(* Schneider Machine Expert - Basic project es1_2pompe_1max_2soglie_scelta_alternanza, file version 3.0.0.0 *)
(* ProjectInformations: Name=New project *)

HARDWARE
  Cpu 0: TM221C40R
  EthernetConfiguration: NetworkName=M221, IpAllocationMode=FixedAddress, IpAddress=0.0.0.0, SubnetMask=0.0.0.0
  SerialLineConfiguration: Baud=Baud19200, Parity=ParityEven, DataBits=DataBits8, StopBits=StopBits1, PhysicalMedium=PhysicalMediumRs485, TransmissionMode=TransmissionModeModbusRtu, SlaveId=1, Addressing=SlaveAddressing
  MastTask: UsePeriodScanMode=false, PeriodScan=100
  FastTask: Period=255
  CpuBehavior: StartingMode=StartAsPreviousState, AutoSaveRamOnEeprom=true, WatchdogPeriod=250

SYMBOLS  (address, symbol, comment, settings)
  %M0       P1_USABILE
  %M1       P2_USABILE
  %M2       P1_SUPERATO_NUMERO_SEC_LAVORATI
  %M3       P2_SUPERATO_NUMERO_SEC_LAVORATI
  %M4       ORA_E_00  "E' mezzanotte?"
  %M5       ALTERNATO_POMPE_GIORNALIERO
  %S6       SB_TB1S  "Time base of 1 s generated by an internal clock"
  %SW51     SW_RTCHHMM  "RTC Function: contains in BCD HHMM: hour and minute"
  %MW0      PROSSIMA_POMPA_CANDIDATA
  %MW1      STRG_ALTERNANZA_ATTUALE
  %TM0      TIMER_POMPA_1  [Preset=10, Base=OneSecond, IsRetentive=true, IsDynamicPreset=true]
  %C0       CONTATORE_P1_SECONDI_LAVORATI  [Preset=0]
  %C1       CONTATORE_P2_SECONDI_LAVORATI  [Preset=0]
  %I0.0     P1_AUTO
  %I0.1     P1_MOTO
  %I0.2     P1_ANOMALIA
  %I0.3     P2_AUTO
  %I0.4     P2_MOTO
  %I0.5     P2_ANOMALIA
  %I0.6     LVL_MIN
  %I0.7     LVL_MAX
  %Q0.0     P1_CMD
  %Q0.1     P2_CMD
  %Q0.2     ERR_STRG_ALTERNANZA_INVALIDA
  %IW0.0    STRG_ALTERNANZA_INPUT  "0 = avvio; 1 = meno ore; 2 = giornaliera semplice;"  [Type=Type_0_10V, Scope=Scope_Normal, Minimum=0, Maximum=1000]

POU New POU
  (* SectionNumber=1 *)

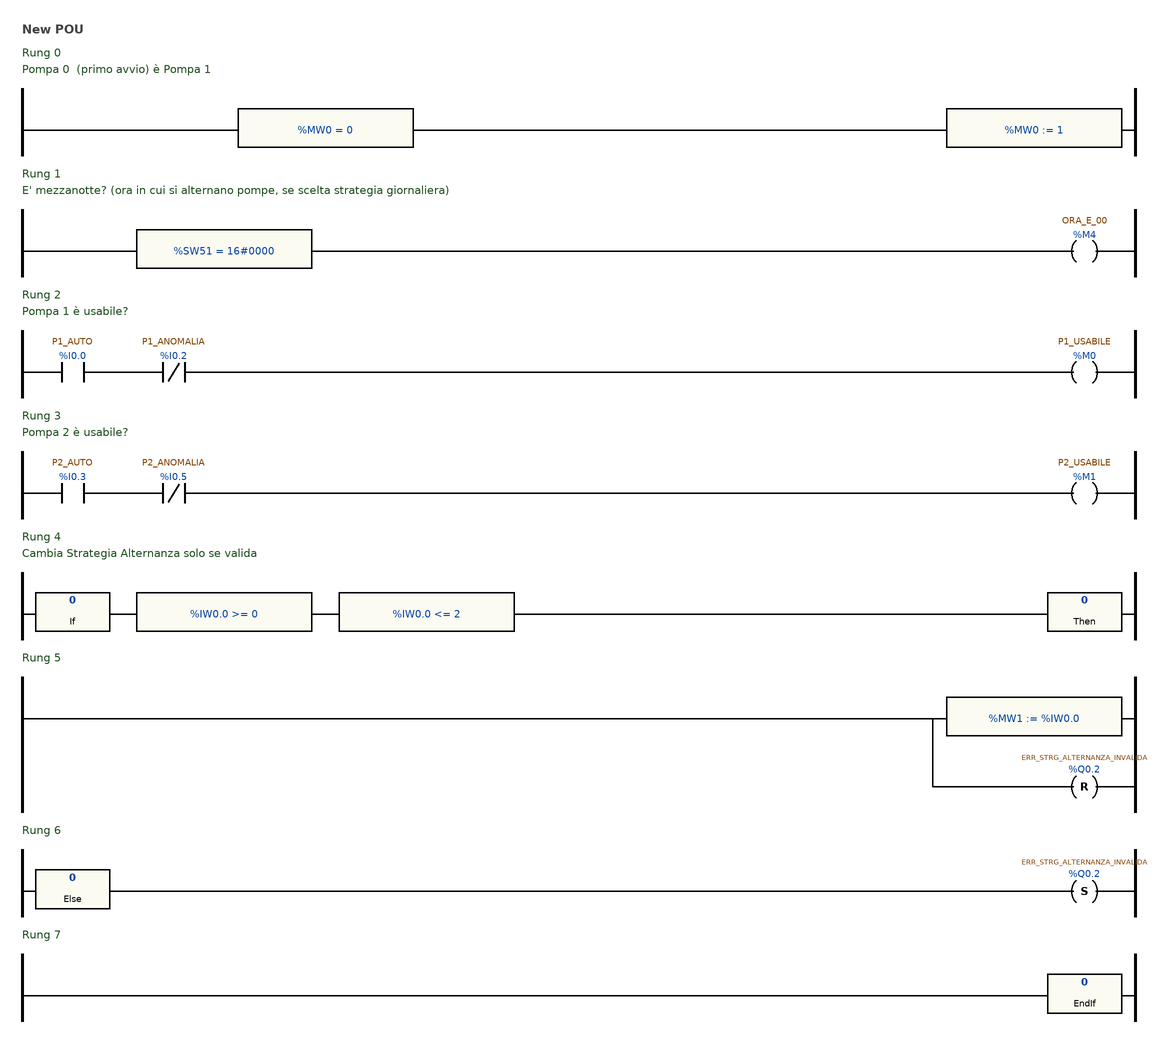

// Rung 0
// Pompa 0  (primo avvio) è Pompa 1
  LD [ %MW0 = 0 ]         (* PROSSIMA_POMPA_CANDIDATA *)
  [ %MW0 := 1 ]           (* PROSSIMA_POMPA_CANDIDATA *)
  // as ST:
  //   IF PROSSIMA_POMPA_CANDIDATA = 0 THEN PROSSIMA_POMPA_CANDIDATA := 1; END_IF;

// Rung 1
// E' mezzanotte? (ora in cui si alternano pompe, se scelta strategia giornaliera)
  LD [ %SW51 = 16#0000 ]  (* SW_RTCHHMM *)
  ST %M4                  (* ORA_E_00 *)
  // as ST:
  //   ORA_E_00 := SW_RTCHHMM = 16#0000;

// Rung 2
// Pompa 1 è usabile?
  LD %I0.0                (* P1_AUTO *)
  ANDN %I0.2              (* P1_ANOMALIA *)
  ST %M0                  (* P1_USABILE *)
  // as ST:
  //   P1_USABILE := P1_AUTO AND NOT P1_ANOMALIA;

// Rung 3
// Pompa 2 è usabile?
  LD %I0.3                (* P2_AUTO *)
  ANDN %I0.5              (* P2_ANOMALIA *)
  ST %M1                  (* P2_USABILE *)
  // as ST:
  //   P2_USABILE := P2_AUTO AND NOT P2_ANOMALIA;

// Rung 4
// Cambia Strategia Alternanza solo se valida
  IF0
  AND [ %IW0.0 >= 0 ]     (* STRG_ALTERNANZA_INPUT *)
  AND [ %IW0.0 <= 2 ]     (* STRG_ALTERNANZA_INPUT *)
  THEN0

// Rung 5
  LD 1
  [ %MW1 := %IW0.0 ]      (* STRG_ALTERNANZA_ATTUALE, STRG_ALTERNANZA_INPUT *)
  R %Q0.2                 (* ERR_STRG_ALTERNANZA_INVALIDA *)
  // as ST:
  //   STRG_ALTERNANZA_ATTUALE := STRG_ALTERNANZA_INPUT;
  //   ERR_STRG_ALTERNANZA_INVALIDA := FALSE;

// Rung 6
  ELSE0
  S %Q0.2                 (* ERR_STRG_ALTERNANZA_INVALIDA *)

// Rung 7
  LD 1
  ENDIF0

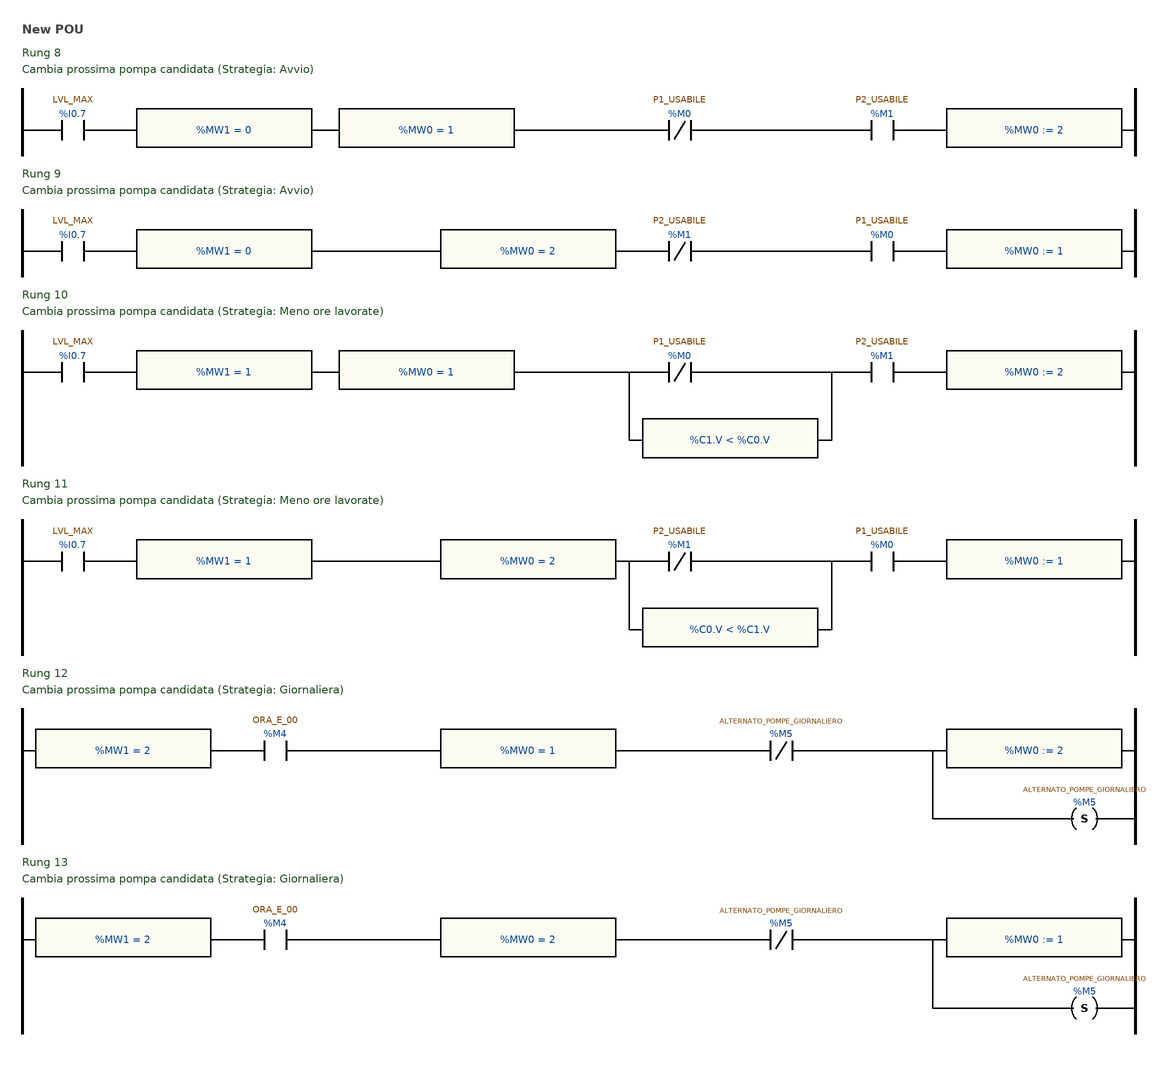

// Rung 8
// Cambia prossima pompa candidata (Strategia: Avvio)
  LD %I0.7                (* LVL_MAX *)
  AND [ %MW1 = 0 ]        (* STRG_ALTERNANZA_ATTUALE *)
  AND [ %MW0 = 1 ]        (* PROSSIMA_POMPA_CANDIDATA *)
  ANDN %M0                (* P1_USABILE *)
  AND %M1                 (* P2_USABILE *)
  [ %MW0 := 2 ]           (* PROSSIMA_POMPA_CANDIDATA *)
  // as ST:
  //   IF LVL_MAX AND STRG_ALTERNANZA_ATTUALE = 0 AND PROSSIMA_POMPA_CANDIDATA = 1 AND NOT P1_USABILE AND P2_USABILE THEN PROSSIMA_POMPA_CANDIDATA := 2; END_IF;

// Rung 9
// Cambia prossima pompa candidata (Strategia: Avvio)
  LD %I0.7                (* LVL_MAX *)
  AND [ %MW1 = 0 ]        (* STRG_ALTERNANZA_ATTUALE *)
  AND [ %MW0 = 2 ]        (* PROSSIMA_POMPA_CANDIDATA *)
  ANDN %M1                (* P2_USABILE *)
  AND %M0                 (* P1_USABILE *)
  [ %MW0 := 1 ]           (* PROSSIMA_POMPA_CANDIDATA *)
  // as ST:
  //   IF LVL_MAX AND STRG_ALTERNANZA_ATTUALE = 0 AND PROSSIMA_POMPA_CANDIDATA = 2 AND NOT P2_USABILE AND P1_USABILE THEN PROSSIMA_POMPA_CANDIDATA := 1; END_IF;

// Rung 10
// Cambia prossima pompa candidata (Strategia: Meno ore lavorate)
  LD %I0.7                (* LVL_MAX *)
  AND [ %MW1 = 1 ]        (* STRG_ALTERNANZA_ATTUALE *)
  AND [ %MW0 = 1 ]        (* PROSSIMA_POMPA_CANDIDATA *)
  AND(N %M0               (* P1_USABILE *)
  OR [ %C1.V < %C0.V ]    (* CONTATORE_P2_SECONDI_LAVORATI, CONTATORE_P1_SECONDI_LAVORATI *)
  )
  AND %M1                 (* P2_USABILE *)
  [ %MW0 := 2 ]           (* PROSSIMA_POMPA_CANDIDATA *)
  // as ST:
  //   IF LVL_MAX AND STRG_ALTERNANZA_ATTUALE = 1 AND PROSSIMA_POMPA_CANDIDATA = 1 AND (NOT P1_USABILE OR CONTATORE_P2_SECONDI_LAVORATI.V < CONTATORE_P1_SECONDI_LAVORATI.V) AND P2_USABILE THEN PROSSIMA_POMPA_CANDIDATA := 2; END_IF;

// Rung 11
// Cambia prossima pompa candidata (Strategia: Meno ore lavorate)
  LD %I0.7                (* LVL_MAX *)
  AND [ %MW1 = 1 ]        (* STRG_ALTERNANZA_ATTUALE *)
  AND [ %MW0 = 2 ]        (* PROSSIMA_POMPA_CANDIDATA *)
  AND(N %M1               (* P2_USABILE *)
  OR [ %C0.V < %C1.V ]    (* CONTATORE_P1_SECONDI_LAVORATI, CONTATORE_P2_SECONDI_LAVORATI *)
  )
  AND %M0                 (* P1_USABILE *)
  [ %MW0 := 1 ]           (* PROSSIMA_POMPA_CANDIDATA *)
  // as ST:
  //   IF LVL_MAX AND STRG_ALTERNANZA_ATTUALE = 1 AND PROSSIMA_POMPA_CANDIDATA = 2 AND (NOT P2_USABILE OR CONTATORE_P1_SECONDI_LAVORATI.V < CONTATORE_P2_SECONDI_LAVORATI.V) AND P1_USABILE THEN PROSSIMA_POMPA_CANDIDATA := 1; END_IF;

// Rung 12
// Cambia prossima pompa candidata (Strategia: Giornaliera)
  LD [ %MW1 = 2 ]         (* STRG_ALTERNANZA_ATTUALE *)
  AND %M4                 (* ORA_E_00 *)
  AND [ %MW0 = 1 ]        (* PROSSIMA_POMPA_CANDIDATA *)
  ANDN %M5                (* ALTERNATO_POMPE_GIORNALIERO *)
  [ %MW0 := 2 ]           (* PROSSIMA_POMPA_CANDIDATA *)
  S %M5                   (* ALTERNATO_POMPE_GIORNALIERO *)
  // as ST:
  //   _t1 := STRG_ALTERNANZA_ATTUALE = 2 AND ORA_E_00 AND PROSSIMA_POMPA_CANDIDATA = 1 AND NOT ALTERNATO_POMPE_GIORNALIERO;
  //   IF _t1 THEN PROSSIMA_POMPA_CANDIDATA := 2; END_IF;
  //   IF _t1 THEN ALTERNATO_POMPE_GIORNALIERO := TRUE; END_IF;

// Rung 13
// Cambia prossima pompa candidata (Strategia: Giornaliera)
  LD [ %MW1 = 2 ]         (* STRG_ALTERNANZA_ATTUALE *)
  AND %M4                 (* ORA_E_00 *)
  AND [ %MW0 = 2 ]        (* PROSSIMA_POMPA_CANDIDATA *)
  ANDN %M5                (* ALTERNATO_POMPE_GIORNALIERO *)
  [ %MW0 := 1 ]           (* PROSSIMA_POMPA_CANDIDATA *)
  S %M5                   (* ALTERNATO_POMPE_GIORNALIERO *)
  // as ST:
  //   _t1 := STRG_ALTERNANZA_ATTUALE = 2 AND ORA_E_00 AND PROSSIMA_POMPA_CANDIDATA = 2 AND NOT ALTERNATO_POMPE_GIORNALIERO;
  //   IF _t1 THEN PROSSIMA_POMPA_CANDIDATA := 1; END_IF;
  //   IF _t1 THEN ALTERNATO_POMPE_GIORNALIERO := TRUE; END_IF;

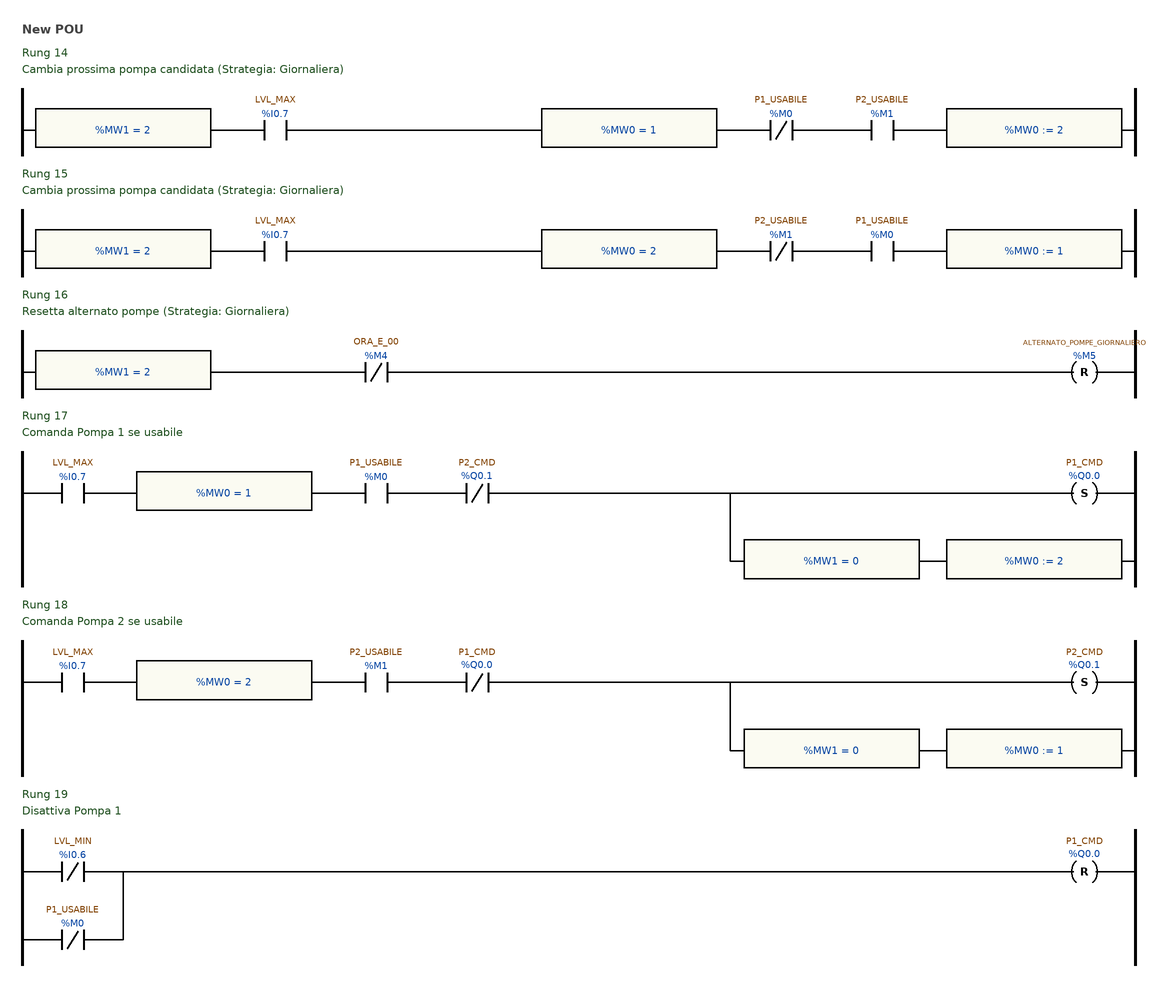

// Rung 14
// Cambia prossima pompa candidata (Strategia: Giornaliera)
  LD [ %MW1 = 2 ]         (* STRG_ALTERNANZA_ATTUALE *)
  AND %I0.7               (* LVL_MAX *)
  AND [ %MW0 = 1 ]        (* PROSSIMA_POMPA_CANDIDATA *)
  ANDN %M0                (* P1_USABILE *)
  AND %M1                 (* P2_USABILE *)
  [ %MW0 := 2 ]           (* PROSSIMA_POMPA_CANDIDATA *)
  // as ST:
  //   IF STRG_ALTERNANZA_ATTUALE = 2 AND LVL_MAX AND PROSSIMA_POMPA_CANDIDATA = 1 AND NOT P1_USABILE AND P2_USABILE THEN PROSSIMA_POMPA_CANDIDATA := 2; END_IF;

// Rung 15
// Cambia prossima pompa candidata (Strategia: Giornaliera)
  LD [ %MW1 = 2 ]         (* STRG_ALTERNANZA_ATTUALE *)
  AND %I0.7               (* LVL_MAX *)
  AND [ %MW0 = 2 ]        (* PROSSIMA_POMPA_CANDIDATA *)
  ANDN %M1                (* P2_USABILE *)
  AND %M0                 (* P1_USABILE *)
  [ %MW0 := 1 ]           (* PROSSIMA_POMPA_CANDIDATA *)
  // as ST:
  //   IF STRG_ALTERNANZA_ATTUALE = 2 AND LVL_MAX AND PROSSIMA_POMPA_CANDIDATA = 2 AND NOT P2_USABILE AND P1_USABILE THEN PROSSIMA_POMPA_CANDIDATA := 1; END_IF;

// Rung 16
// Resetta alternato pompe (Strategia: Giornaliera)
  LD [ %MW1 = 2 ]         (* STRG_ALTERNANZA_ATTUALE *)
  ANDN %M4                (* ORA_E_00 *)
  R %M5                   (* ALTERNATO_POMPE_GIORNALIERO *)
  // as ST:
  //   IF STRG_ALTERNANZA_ATTUALE = 2 AND NOT ORA_E_00 THEN ALTERNATO_POMPE_GIORNALIERO := FALSE; END_IF;

// Rung 17
// Comanda Pompa 1 se usabile
  LD %I0.7                (* LVL_MAX *)
  AND [ %MW0 = 1 ]        (* PROSSIMA_POMPA_CANDIDATA *)
  AND %M0                 (* P1_USABILE *)
  ANDN %Q0.1              (* P2_CMD *)
  MPS
  S %Q0.0                 (* P1_CMD *)
  MPP
  AND [ %MW1 = 0 ]        (* STRG_ALTERNANZA_ATTUALE *)
  [ %MW0 := 2 ]           (* PROSSIMA_POMPA_CANDIDATA *)
  // as ST:
  //   IF LVL_MAX AND PROSSIMA_POMPA_CANDIDATA = 1 AND P1_USABILE AND NOT P2_CMD THEN P1_CMD := TRUE; END_IF;
  //   IF LVL_MAX AND PROSSIMA_POMPA_CANDIDATA = 1 AND P1_USABILE AND NOT P2_CMD AND STRG_ALTERNANZA_ATTUALE = 0 THEN PROSSIMA_POMPA_CANDIDATA := 2; END_IF;

// Rung 18
// Comanda Pompa 2 se usabile
  LD %I0.7                (* LVL_MAX *)
  AND [ %MW0 = 2 ]        (* PROSSIMA_POMPA_CANDIDATA *)
  AND %M1                 (* P2_USABILE *)
  ANDN %Q0.0              (* P1_CMD *)
  MPS
  S %Q0.1                 (* P2_CMD *)
  MPP
  AND [ %MW1 = 0 ]        (* STRG_ALTERNANZA_ATTUALE *)
  [ %MW0 := 1 ]           (* PROSSIMA_POMPA_CANDIDATA *)
  // as ST:
  //   IF LVL_MAX AND PROSSIMA_POMPA_CANDIDATA = 2 AND P2_USABILE AND NOT P1_CMD THEN P2_CMD := TRUE; END_IF;
  //   IF LVL_MAX AND PROSSIMA_POMPA_CANDIDATA = 2 AND P2_USABILE AND NOT P1_CMD AND STRG_ALTERNANZA_ATTUALE = 0 THEN PROSSIMA_POMPA_CANDIDATA := 1; END_IF;

// Rung 19
// Disattiva Pompa 1
  LDN %I0.6               (* LVL_MIN *)
  ORN %M0                 (* P1_USABILE *)
  R %Q0.0                 (* P1_CMD *)
  // as ST:
  //   IF NOT LVL_MIN OR NOT P1_USABILE THEN P1_CMD := FALSE; END_IF;

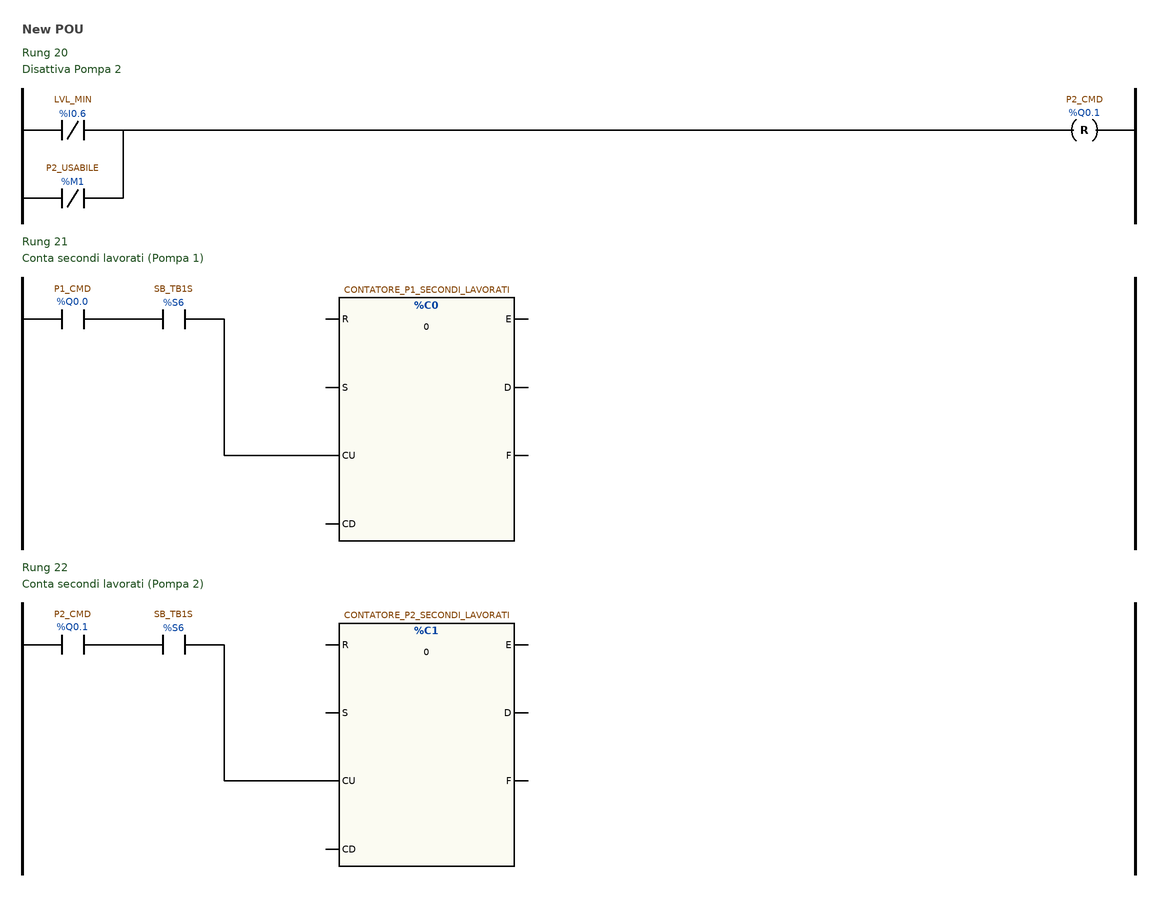

// Rung 20
// Disattiva Pompa 2
  LDN %I0.6               (* LVL_MIN *)
  ORN %M1                 (* P2_USABILE *)
  R %Q0.1                 (* P2_CMD *)
  // as ST:
  //   IF NOT LVL_MIN OR NOT P2_USABILE THEN P2_CMD := FALSE; END_IF;

// Rung 21
// Conta secondi lavorati (Pompa 1)
  BLK %C0                 (* CONTATORE_P1_SECONDI_LAVORATI *)
  LD %Q0.0                (* P1_CMD *)
  AND %S6                 (* SB_TB1S *)
  CU
  END_BLK
  // as ST:
  //   CONTATORE_P1_SECONDI_LAVORATI(CU := P1_CMD AND SB_TB1S);

// Rung 22
// Conta secondi lavorati (Pompa 2)
  BLK %C1                 (* CONTATORE_P2_SECONDI_LAVORATI *)
  LD %Q0.1                (* P2_CMD *)
  AND %S6                 (* SB_TB1S *)
  CU
  END_BLK
  // as ST:
  //   CONTATORE_P2_SECONDI_LAVORATI(CU := P2_CMD AND SB_TB1S);
